Fanuc TP program (LS listing): RECSTEPB.LS

/PROG  RECSTEPB
/ATTR
OWNER		= MNEDITOR;
COMMENT		= "RecStepB";
PROG_SIZE	= 0;
CREATE		= DATE 26-01-01  TIME 00:00:00;
MODIFIED	= DATE 26-01-01  TIME 00:00:00;
FILE_NAME	= ;
VERSION		= 0;
LINE_COUNT	= 6;
MEMORY_SIZE	= 0;
PROTECT		= READ_WRITE;
TCD:  STACK_SIZE	= 0,
      TASK_PRIORITY	= 50,
      TIME_SLICE	= 0,
      BUSY_LAMP_OFF	= 0,
      ABORT_REQUEST	= 0,
      PAUSE_REQUEST	= 0;
DEFAULT_GROUP	= 1,*,*,*,*;
CONTROL_CODE	= 00000000 00000000;
/MN
   1:  !RAPID RecordProbe.RecStepB ;
   2:  IF (R[2:recCtrl.state]=1) THEN ;
   3:  R[2:recCtrl.state]=2    ;
   4:  R[1:recCtrl.counter]=R[1:recCtrl.counter]+10    ;
   5:  ENDIF ;
   6:  F[1]=(OFF) ;
/POS
/END
